// TIA Portal V17 export
// export: Created 2023-12-22T15:05:24.7176583Z, ExportSetting WithDefaults, DisplayName Totally Integrated Automation Portal, DisplayVersion V17, DisplayName TIA Portal Openness, DisplayVersion V17, DisplayName TIA Portal Version Control Interface, DisplayVersion V17, DisplayName STEP 7 Professional, DisplayVersion V17, DisplayName STEP 7 Safety, DisplayVersion V17, DisplayName WinCC Advanced, DisplayVersion V17
FUNCTION "Line_Alarms" : Void   // FC3, LAD
{ S7_Optimized_Access := 'TRUE' }
VERSION : 0.1
// stored: AutoNumber true, IsIECCheckEnabled false, SetENOAutomatically false, UDAEnableTagReadback false
   VAR_INPUT
      All_Lines : Int;   // Кол-во линий
   END_VAR
   VAR_IN_OUT
      Alm_REQ : Int;   // Запрос аварии
      Alm_Now : Int;   // Авария сейчас
      Ready : Bool;   // Готовность
   END_VAR
   VAR_TEMP   // added for the SCL form of the ladder/FBD networks
      _w1 : Bool;
      _w2 : Bool;
      _w3 : Bool;
      _w4 : Bool;
      _w5 : Bool;
      _w6 : Bool;
      _w7 : Bool;
   END_VAR
BEGIN

REGION Network 1: Проверка корректности выбранной линии
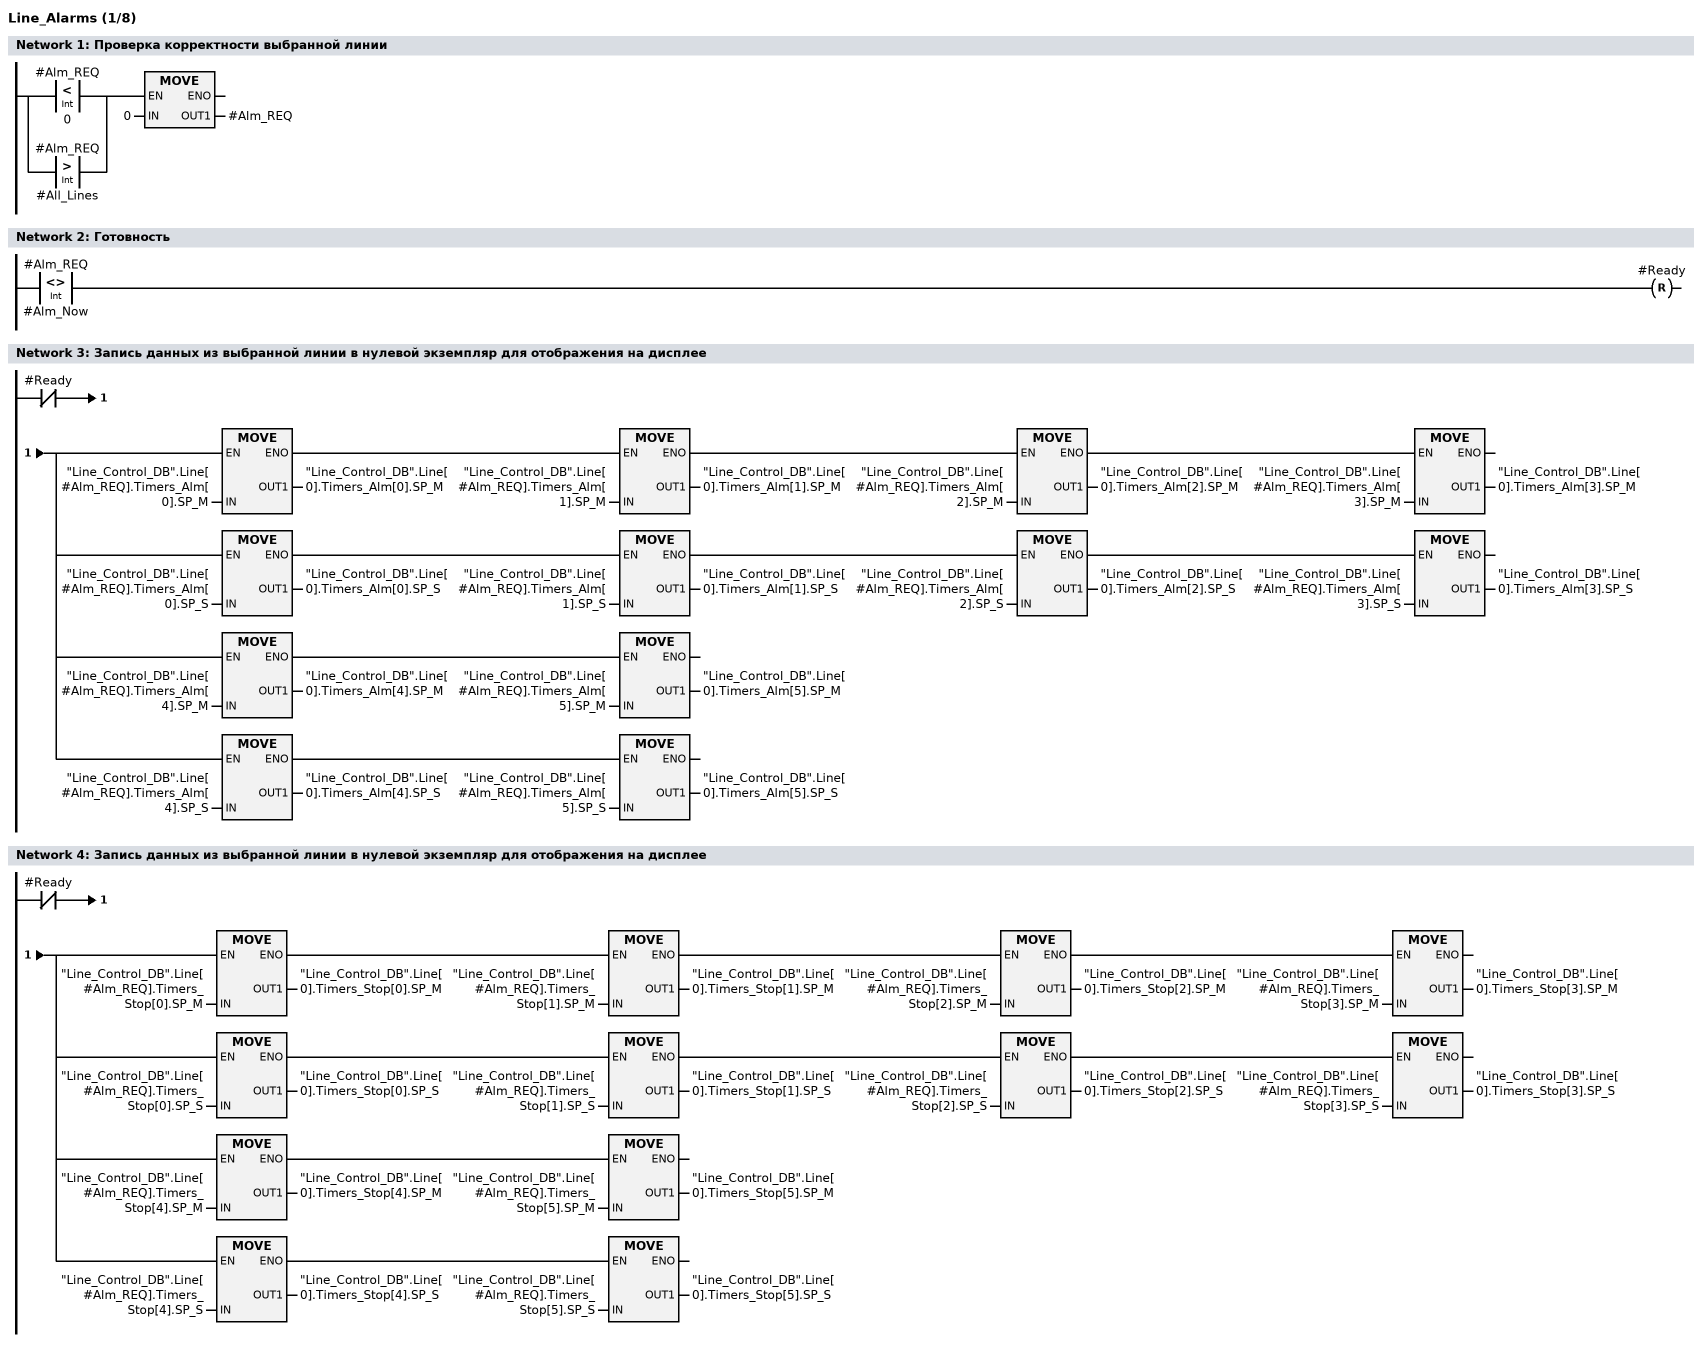
   RUNG wire#powerrail
      { S7_Templates := "SrcType := Int" } LT_Contact(in1 := #Alm_REQ, in2 := 0)
      wire#w1
      Move(in := 0, out1 => #Alm_REQ)
   END_RUNG
   RUNG wire#powerrail
      { S7_Templates := "SrcType := Int" } GT_Contact(in1 := #Alm_REQ, in2 := #All_Lines)
   END_RUNG wire#w1
   // the same network as SCL:
   IF (#Alm_REQ < 0) OR (#Alm_REQ > #All_Lines) THEN #Alm_REQ := 0; END_IF;
END_REGION

REGION Network 2: Готовность
   RUNG wire#powerrail
      { S7_Templates := "SrcType := Int" } NE_Contact(in1 := #Alm_REQ, in2 := #Alm_Now)
      R_Coil( #Ready )
   END_RUNG
   // the same network as SCL:
   IF #Alm_REQ <> #Alm_Now THEN #Ready := FALSE; END_IF;
END_REGION

REGION Network 3: Запись данных из выбранной линии в нулевой экземпляр для отображения на дисплее
   RUNG wire#powerrail
      I_Contact( #Ready )
      wire#w1
      Move(in := "Line_Control_DB".Line[#Alm_REQ].Timers_Alm[0].SP_M, out1 => "Line_Control_DB".Line[0].Timers_Alm[0].SP_M)
      Move(in := "Line_Control_DB".Line[#Alm_REQ].Timers_Alm[1].SP_M, out1 => "Line_Control_DB".Line[0].Timers_Alm[1].SP_M)
      Move(in := "Line_Control_DB".Line[#Alm_REQ].Timers_Alm[2].SP_M, out1 => "Line_Control_DB".Line[0].Timers_Alm[2].SP_M)
      Move(in := "Line_Control_DB".Line[#Alm_REQ].Timers_Alm[3].SP_M, out1 => "Line_Control_DB".Line[0].Timers_Alm[3].SP_M)
   END_RUNG
   RUNG wire#w1
      Move(in := "Line_Control_DB".Line[#Alm_REQ].Timers_Alm[0].SP_S, out1 => "Line_Control_DB".Line[0].Timers_Alm[0].SP_S)
      Move(in := "Line_Control_DB".Line[#Alm_REQ].Timers_Alm[1].SP_S, out1 => "Line_Control_DB".Line[0].Timers_Alm[1].SP_S)
      Move(in := "Line_Control_DB".Line[#Alm_REQ].Timers_Alm[2].SP_S, out1 => "Line_Control_DB".Line[0].Timers_Alm[2].SP_S)
      Move(in := "Line_Control_DB".Line[#Alm_REQ].Timers_Alm[3].SP_S, out1 => "Line_Control_DB".Line[0].Timers_Alm[3].SP_S)
   END_RUNG
   RUNG wire#w1
      Move(in := "Line_Control_DB".Line[#Alm_REQ].Timers_Alm[4].SP_M, out1 => "Line_Control_DB".Line[0].Timers_Alm[4].SP_M)
      Move(in := "Line_Control_DB".Line[#Alm_REQ].Timers_Alm[5].SP_M, out1 => "Line_Control_DB".Line[0].Timers_Alm[5].SP_M)
   END_RUNG
   RUNG wire#w1
      Move(in := "Line_Control_DB".Line[#Alm_REQ].Timers_Alm[4].SP_S, out1 => "Line_Control_DB".Line[0].Timers_Alm[4].SP_S)
      Move(in := "Line_Control_DB".Line[#Alm_REQ].Timers_Alm[5].SP_S, out1 => "Line_Control_DB".Line[0].Timers_Alm[5].SP_S)
   END_RUNG
   // the same network as SCL:
   IF NOT #Ready THEN
       "Line_Control_DB".Line[0].Timers_Alm[0].SP_M := "Line_Control_DB".Line[#Alm_REQ].Timers_Alm[0].SP_M;
       "Line_Control_DB".Line[0].Timers_Alm[1].SP_M := "Line_Control_DB".Line[#Alm_REQ].Timers_Alm[1].SP_M;
       "Line_Control_DB".Line[0].Timers_Alm[2].SP_M := "Line_Control_DB".Line[#Alm_REQ].Timers_Alm[2].SP_M;
       "Line_Control_DB".Line[0].Timers_Alm[3].SP_M := "Line_Control_DB".Line[#Alm_REQ].Timers_Alm[3].SP_M;
       "Line_Control_DB".Line[0].Timers_Alm[0].SP_S := "Line_Control_DB".Line[#Alm_REQ].Timers_Alm[0].SP_S;
       "Line_Control_DB".Line[0].Timers_Alm[1].SP_S := "Line_Control_DB".Line[#Alm_REQ].Timers_Alm[1].SP_S;
       "Line_Control_DB".Line[0].Timers_Alm[2].SP_S := "Line_Control_DB".Line[#Alm_REQ].Timers_Alm[2].SP_S;
       "Line_Control_DB".Line[0].Timers_Alm[3].SP_S := "Line_Control_DB".Line[#Alm_REQ].Timers_Alm[3].SP_S;
       "Line_Control_DB".Line[0].Timers_Alm[4].SP_M := "Line_Control_DB".Line[#Alm_REQ].Timers_Alm[4].SP_M;
       "Line_Control_DB".Line[0].Timers_Alm[5].SP_M := "Line_Control_DB".Line[#Alm_REQ].Timers_Alm[5].SP_M;
       "Line_Control_DB".Line[0].Timers_Alm[4].SP_S := "Line_Control_DB".Line[#Alm_REQ].Timers_Alm[4].SP_S;
       "Line_Control_DB".Line[0].Timers_Alm[5].SP_S := "Line_Control_DB".Line[#Alm_REQ].Timers_Alm[5].SP_S;
   END_IF;
END_REGION

REGION Network 4: Запись данных из выбранной линии в нулевой экземпляр для отображения на дисплее
   RUNG wire#powerrail
      I_Contact( #Ready )
      wire#w1
      Move(in := "Line_Control_DB".Line[#Alm_REQ].Timers_Stop[0].SP_M, out1 => "Line_Control_DB".Line[0].Timers_Stop[0].SP_M)
      Move(in := "Line_Control_DB".Line[#Alm_REQ].Timers_Stop[1].SP_M, out1 => "Line_Control_DB".Line[0].Timers_Stop[1].SP_M)
      Move(in := "Line_Control_DB".Line[#Alm_REQ].Timers_Stop[2].SP_M, out1 => "Line_Control_DB".Line[0].Timers_Stop[2].SP_M)
      Move(in := "Line_Control_DB".Line[#Alm_REQ].Timers_Stop[3].SP_M, out1 => "Line_Control_DB".Line[0].Timers_Stop[3].SP_M)
   END_RUNG
   RUNG wire#w1
      Move(in := "Line_Control_DB".Line[#Alm_REQ].Timers_Stop[0].SP_S, out1 => "Line_Control_DB".Line[0].Timers_Stop[0].SP_S)
      Move(in := "Line_Control_DB".Line[#Alm_REQ].Timers_Stop[1].SP_S, out1 => "Line_Control_DB".Line[0].Timers_Stop[1].SP_S)
      Move(in := "Line_Control_DB".Line[#Alm_REQ].Timers_Stop[2].SP_S, out1 => "Line_Control_DB".Line[0].Timers_Stop[2].SP_S)
      Move(in := "Line_Control_DB".Line[#Alm_REQ].Timers_Stop[3].SP_S, out1 => "Line_Control_DB".Line[0].Timers_Stop[3].SP_S)
   END_RUNG
   RUNG wire#w1
      Move(in := "Line_Control_DB".Line[#Alm_REQ].Timers_Stop[4].SP_M, out1 => "Line_Control_DB".Line[0].Timers_Stop[4].SP_M)
      Move(in := "Line_Control_DB".Line[#Alm_REQ].Timers_Stop[5].SP_M, out1 => "Line_Control_DB".Line[0].Timers_Stop[5].SP_M)
   END_RUNG
   RUNG wire#w1
      Move(in := "Line_Control_DB".Line[#Alm_REQ].Timers_Stop[4].SP_S, out1 => "Line_Control_DB".Line[0].Timers_Stop[4].SP_S)
      Move(in := "Line_Control_DB".Line[#Alm_REQ].Timers_Stop[5].SP_S, out1 => "Line_Control_DB".Line[0].Timers_Stop[5].SP_S)
   END_RUNG
   // the same network as SCL:
   IF NOT #Ready THEN
       "Line_Control_DB".Line[0].Timers_Stop[0].SP_M := "Line_Control_DB".Line[#Alm_REQ].Timers_Stop[0].SP_M;
       "Line_Control_DB".Line[0].Timers_Stop[1].SP_M := "Line_Control_DB".Line[#Alm_REQ].Timers_Stop[1].SP_M;
       "Line_Control_DB".Line[0].Timers_Stop[2].SP_M := "Line_Control_DB".Line[#Alm_REQ].Timers_Stop[2].SP_M;
       "Line_Control_DB".Line[0].Timers_Stop[3].SP_M := "Line_Control_DB".Line[#Alm_REQ].Timers_Stop[3].SP_M;
       "Line_Control_DB".Line[0].Timers_Stop[0].SP_S := "Line_Control_DB".Line[#Alm_REQ].Timers_Stop[0].SP_S;
       "Line_Control_DB".Line[0].Timers_Stop[1].SP_S := "Line_Control_DB".Line[#Alm_REQ].Timers_Stop[1].SP_S;
       "Line_Control_DB".Line[0].Timers_Stop[2].SP_S := "Line_Control_DB".Line[#Alm_REQ].Timers_Stop[2].SP_S;
       "Line_Control_DB".Line[0].Timers_Stop[3].SP_S := "Line_Control_DB".Line[#Alm_REQ].Timers_Stop[3].SP_S;
       "Line_Control_DB".Line[0].Timers_Stop[4].SP_M := "Line_Control_DB".Line[#Alm_REQ].Timers_Stop[4].SP_M;
       "Line_Control_DB".Line[0].Timers_Stop[5].SP_M := "Line_Control_DB".Line[#Alm_REQ].Timers_Stop[5].SP_M;
       "Line_Control_DB".Line[0].Timers_Stop[4].SP_S := "Line_Control_DB".Line[#Alm_REQ].Timers_Stop[4].SP_S;
       "Line_Control_DB".Line[0].Timers_Stop[5].SP_S := "Line_Control_DB".Line[#Alm_REQ].Timers_Stop[5].SP_S;
   END_IF;
END_REGION

REGION Network 5: Запись данных из выбранной линии в нулевой экземпляр для отображения на дисплее
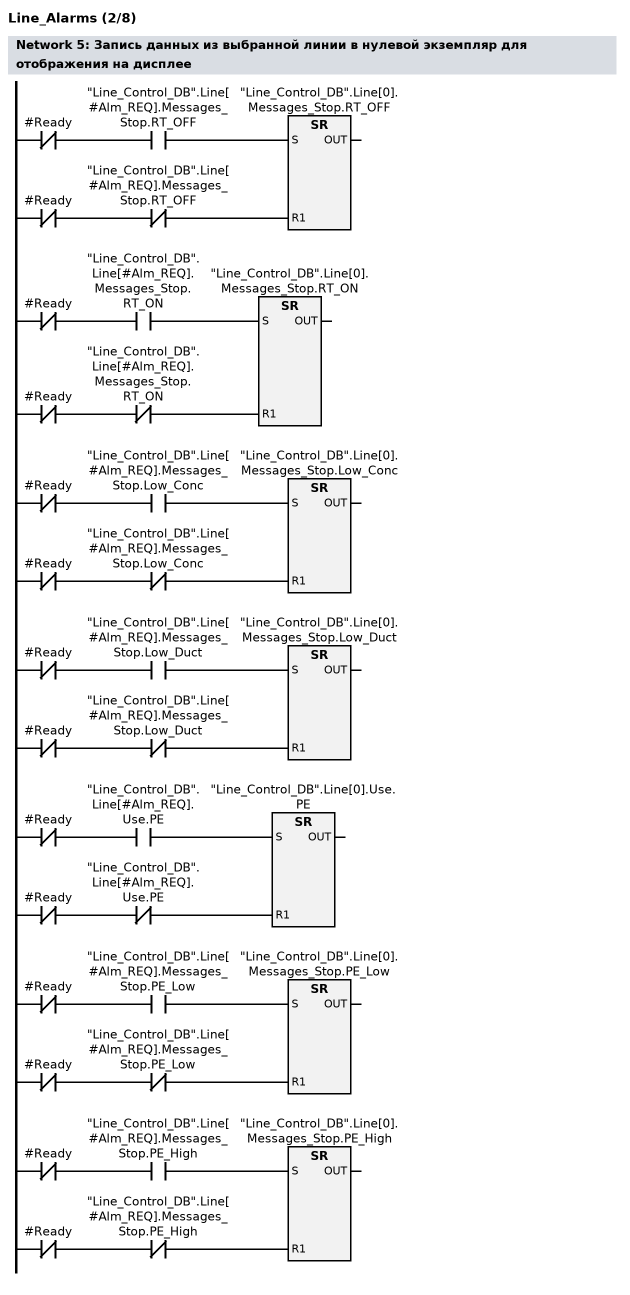
   RUNG wire#powerrail
      I_Contact( #Ready )
      Contact( "Line_Control_DB".Line[#Alm_REQ].Messages_Stop.RT_OFF )
      S_SR(operand := "Line_Control_DB".Line[0].Messages_Stop.RT_OFF, r1 := wire#w1)
   END_RUNG
   RUNG wire#powerrail
      I_Contact( #Ready )
      I_Contact( "Line_Control_DB".Line[#Alm_REQ].Messages_Stop.RT_OFF )
   END_RUNG wire#w1
   RUNG wire#powerrail
      I_Contact( #Ready )
      Contact( "Line_Control_DB".Line[#Alm_REQ].Messages_Stop.RT_ON )
      S_SR(operand := "Line_Control_DB".Line[0].Messages_Stop.RT_ON, r1 := wire#w2)
   END_RUNG
   RUNG wire#powerrail
      I_Contact( #Ready )
      I_Contact( "Line_Control_DB".Line[#Alm_REQ].Messages_Stop.RT_ON )
   END_RUNG wire#w2
   RUNG wire#powerrail
      I_Contact( #Ready )
      Contact( "Line_Control_DB".Line[#Alm_REQ].Messages_Stop.Low_Conc )
      S_SR(operand := "Line_Control_DB".Line[0].Messages_Stop.Low_Conc, r1 := wire#w3)
   END_RUNG
   RUNG wire#powerrail
      I_Contact( #Ready )
      I_Contact( "Line_Control_DB".Line[#Alm_REQ].Messages_Stop.Low_Conc )
   END_RUNG wire#w3
   RUNG wire#powerrail
      I_Contact( #Ready )
      Contact( "Line_Control_DB".Line[#Alm_REQ].Messages_Stop.Low_Duct )
      S_SR(operand := "Line_Control_DB".Line[0].Messages_Stop.Low_Duct, r1 := wire#w4)
   END_RUNG
   RUNG wire#powerrail
      I_Contact( #Ready )
      I_Contact( "Line_Control_DB".Line[#Alm_REQ].Messages_Stop.Low_Duct )
   END_RUNG wire#w4
   RUNG wire#powerrail
      I_Contact( #Ready )
      Contact( "Line_Control_DB".Line[#Alm_REQ].Use.PE )
      S_SR(operand := "Line_Control_DB".Line[0].Use.PE, r1 := wire#w5)
   END_RUNG
   RUNG wire#powerrail
      I_Contact( #Ready )
      I_Contact( "Line_Control_DB".Line[#Alm_REQ].Use.PE )
   END_RUNG wire#w5
   RUNG wire#powerrail
      I_Contact( #Ready )
      Contact( "Line_Control_DB".Line[#Alm_REQ].Messages_Stop.PE_Low )
      S_SR(operand := "Line_Control_DB".Line[0].Messages_Stop.PE_Low, r1 := wire#w6)
   END_RUNG
   RUNG wire#powerrail
      I_Contact( #Ready )
      I_Contact( "Line_Control_DB".Line[#Alm_REQ].Messages_Stop.PE_Low )
   END_RUNG wire#w6
   RUNG wire#powerrail
      I_Contact( #Ready )
      Contact( "Line_Control_DB".Line[#Alm_REQ].Messages_Stop.PE_High )
      S_SR(operand := "Line_Control_DB".Line[0].Messages_Stop.PE_High, r1 := wire#w7)
   END_RUNG
   RUNG wire#powerrail
      I_Contact( #Ready )
      I_Contact( "Line_Control_DB".Line[#Alm_REQ].Messages_Stop.PE_High )
   END_RUNG wire#w7
   // the same network as SCL:
   #_w1 := NOT #Ready AND NOT "Line_Control_DB".Line[#Alm_REQ].Messages_Stop.RT_OFF;
   IF NOT #Ready AND "Line_Control_DB".Line[#Alm_REQ].Messages_Stop.RT_OFF THEN
       "Line_Control_DB".Line[0].Messages_Stop.RT_OFF := TRUE;   // SR flip-flop
   END_IF;
   IF #_w1 THEN "Line_Control_DB".Line[0].Messages_Stop.RT_OFF := FALSE; END_IF;
   #_w2 := NOT #Ready AND NOT "Line_Control_DB".Line[#Alm_REQ].Messages_Stop.RT_ON;
   IF NOT #Ready AND "Line_Control_DB".Line[#Alm_REQ].Messages_Stop.RT_ON THEN
       "Line_Control_DB".Line[0].Messages_Stop.RT_ON := TRUE;   // SR flip-flop
   END_IF;
   IF #_w2 THEN "Line_Control_DB".Line[0].Messages_Stop.RT_ON := FALSE; END_IF;
   #_w3 := NOT #Ready AND NOT "Line_Control_DB".Line[#Alm_REQ].Messages_Stop.Low_Conc;
   IF NOT #Ready AND "Line_Control_DB".Line[#Alm_REQ].Messages_Stop.Low_Conc THEN
       "Line_Control_DB".Line[0].Messages_Stop.Low_Conc := TRUE;   // SR flip-flop
   END_IF;
   IF #_w3 THEN "Line_Control_DB".Line[0].Messages_Stop.Low_Conc := FALSE; END_IF;
   #_w4 := NOT #Ready AND NOT "Line_Control_DB".Line[#Alm_REQ].Messages_Stop.Low_Duct;
   IF NOT #Ready AND "Line_Control_DB".Line[#Alm_REQ].Messages_Stop.Low_Duct THEN
       "Line_Control_DB".Line[0].Messages_Stop.Low_Duct := TRUE;   // SR flip-flop
   END_IF;
   IF #_w4 THEN "Line_Control_DB".Line[0].Messages_Stop.Low_Duct := FALSE; END_IF;
   #_w5 := NOT #Ready AND NOT "Line_Control_DB".Line[#Alm_REQ].Use.PE;
   IF NOT #Ready AND "Line_Control_DB".Line[#Alm_REQ].Use.PE THEN
       "Line_Control_DB".Line[0].Use.PE := TRUE;   // SR flip-flop
   END_IF;
   IF #_w5 THEN "Line_Control_DB".Line[0].Use.PE := FALSE; END_IF;
   #_w6 := NOT #Ready AND NOT "Line_Control_DB".Line[#Alm_REQ].Messages_Stop.PE_Low;
   IF NOT #Ready AND "Line_Control_DB".Line[#Alm_REQ].Messages_Stop.PE_Low THEN
       "Line_Control_DB".Line[0].Messages_Stop.PE_Low := TRUE;   // SR flip-flop
   END_IF;
   IF #_w6 THEN "Line_Control_DB".Line[0].Messages_Stop.PE_Low := FALSE; END_IF;
   #_w7 := NOT #Ready AND NOT "Line_Control_DB".Line[#Alm_REQ].Messages_Stop.PE_High;
   IF NOT #Ready AND "Line_Control_DB".Line[#Alm_REQ].Messages_Stop.PE_High THEN
       "Line_Control_DB".Line[0].Messages_Stop.PE_High := TRUE;   // SR flip-flop
   END_IF;
   IF #_w7 THEN "Line_Control_DB".Line[0].Messages_Stop.PE_High := FALSE; END_IF;
END_REGION

REGION Network 6: Запись данных из выбранной линии в нулевой экземпляр для отображения на дисплее
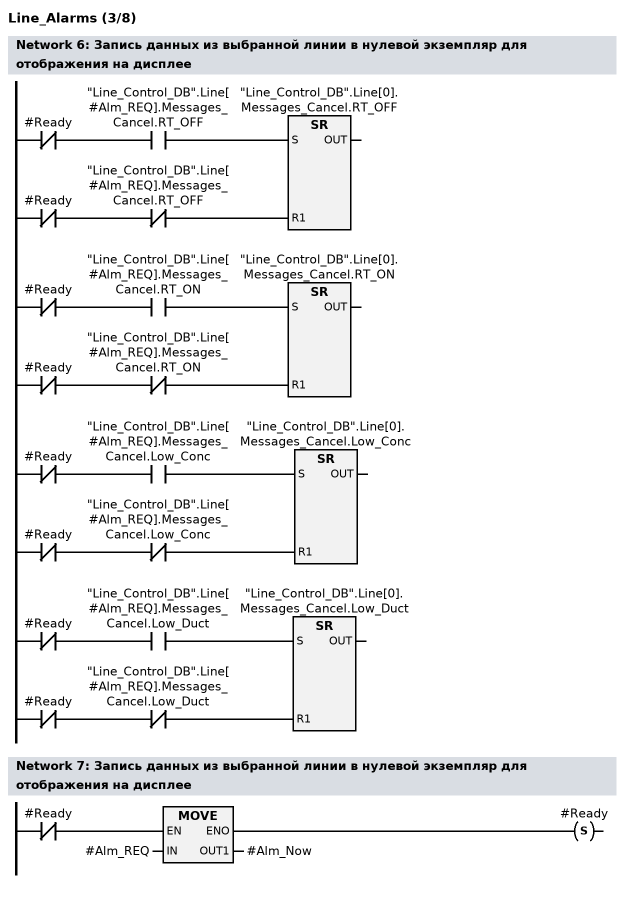
   RUNG wire#powerrail
      I_Contact( #Ready )
      Contact( "Line_Control_DB".Line[#Alm_REQ].Messages_Cancel.RT_OFF )
      S_SR(operand := "Line_Control_DB".Line[0].Messages_Cancel.RT_OFF, r1 := wire#w1)
   END_RUNG
   RUNG wire#powerrail
      I_Contact( #Ready )
      I_Contact( "Line_Control_DB".Line[#Alm_REQ].Messages_Cancel.RT_OFF )
   END_RUNG wire#w1
   RUNG wire#powerrail
      I_Contact( #Ready )
      Contact( "Line_Control_DB".Line[#Alm_REQ].Messages_Cancel.RT_ON )
      S_SR(operand := "Line_Control_DB".Line[0].Messages_Cancel.RT_ON, r1 := wire#w2)
   END_RUNG
   RUNG wire#powerrail
      I_Contact( #Ready )
      I_Contact( "Line_Control_DB".Line[#Alm_REQ].Messages_Cancel.RT_ON )
   END_RUNG wire#w2
   RUNG wire#powerrail
      I_Contact( #Ready )
      Contact( "Line_Control_DB".Line[#Alm_REQ].Messages_Cancel.Low_Conc )
      S_SR(operand := "Line_Control_DB".Line[0].Messages_Cancel.Low_Conc, r1 := wire#w3)
   END_RUNG
   RUNG wire#powerrail
      I_Contact( #Ready )
      I_Contact( "Line_Control_DB".Line[#Alm_REQ].Messages_Cancel.Low_Conc )
   END_RUNG wire#w3
   RUNG wire#powerrail
      I_Contact( #Ready )
      Contact( "Line_Control_DB".Line[#Alm_REQ].Messages_Cancel.Low_Duct )
      S_SR(operand := "Line_Control_DB".Line[0].Messages_Cancel.Low_Duct, r1 := wire#w4)
   END_RUNG
   RUNG wire#powerrail
      I_Contact( #Ready )
      I_Contact( "Line_Control_DB".Line[#Alm_REQ].Messages_Cancel.Low_Duct )
   END_RUNG wire#w4
   // the same network as SCL:
   #_w1 := NOT #Ready AND NOT "Line_Control_DB".Line[#Alm_REQ].Messages_Cancel.RT_OFF;
   IF NOT #Ready AND "Line_Control_DB".Line[#Alm_REQ].Messages_Cancel.RT_OFF THEN
       "Line_Control_DB".Line[0].Messages_Cancel.RT_OFF := TRUE;   // SR flip-flop
   END_IF;
   IF #_w1 THEN "Line_Control_DB".Line[0].Messages_Cancel.RT_OFF := FALSE; END_IF;
   #_w2 := NOT #Ready AND NOT "Line_Control_DB".Line[#Alm_REQ].Messages_Cancel.RT_ON;
   IF NOT #Ready AND "Line_Control_DB".Line[#Alm_REQ].Messages_Cancel.RT_ON THEN
       "Line_Control_DB".Line[0].Messages_Cancel.RT_ON := TRUE;   // SR flip-flop
   END_IF;
   IF #_w2 THEN "Line_Control_DB".Line[0].Messages_Cancel.RT_ON := FALSE; END_IF;
   #_w3 := NOT #Ready AND NOT "Line_Control_DB".Line[#Alm_REQ].Messages_Cancel.Low_Conc;
   IF NOT #Ready AND "Line_Control_DB".Line[#Alm_REQ].Messages_Cancel.Low_Conc THEN
       "Line_Control_DB".Line[0].Messages_Cancel.Low_Conc := TRUE;   // SR flip-flop
   END_IF;
   IF #_w3 THEN "Line_Control_DB".Line[0].Messages_Cancel.Low_Conc := FALSE; END_IF;
   #_w4 := NOT #Ready AND NOT "Line_Control_DB".Line[#Alm_REQ].Messages_Cancel.Low_Duct;
   IF NOT #Ready AND "Line_Control_DB".Line[#Alm_REQ].Messages_Cancel.Low_Duct THEN
       "Line_Control_DB".Line[0].Messages_Cancel.Low_Duct := TRUE;   // SR flip-flop
   END_IF;
   IF #_w4 THEN "Line_Control_DB".Line[0].Messages_Cancel.Low_Duct := FALSE; END_IF;
END_REGION

REGION Network 7: Запись данных из выбранной линии в нулевой экземпляр для отображения на дисплее
   RUNG wire#powerrail
      I_Contact( #Ready )
      Move(in := #Alm_REQ, out1 => #Alm_Now)
      S_Coil( #Ready )
   END_RUNG
   // the same network as SCL:
   IF NOT #Ready THEN
       #Alm_Now := #Alm_REQ;
       #Ready := TRUE;
   END_IF;
END_REGION

REGION Network 8: Запись данных из выбранной линии в нулевой экземпляр для отображения на дисплее
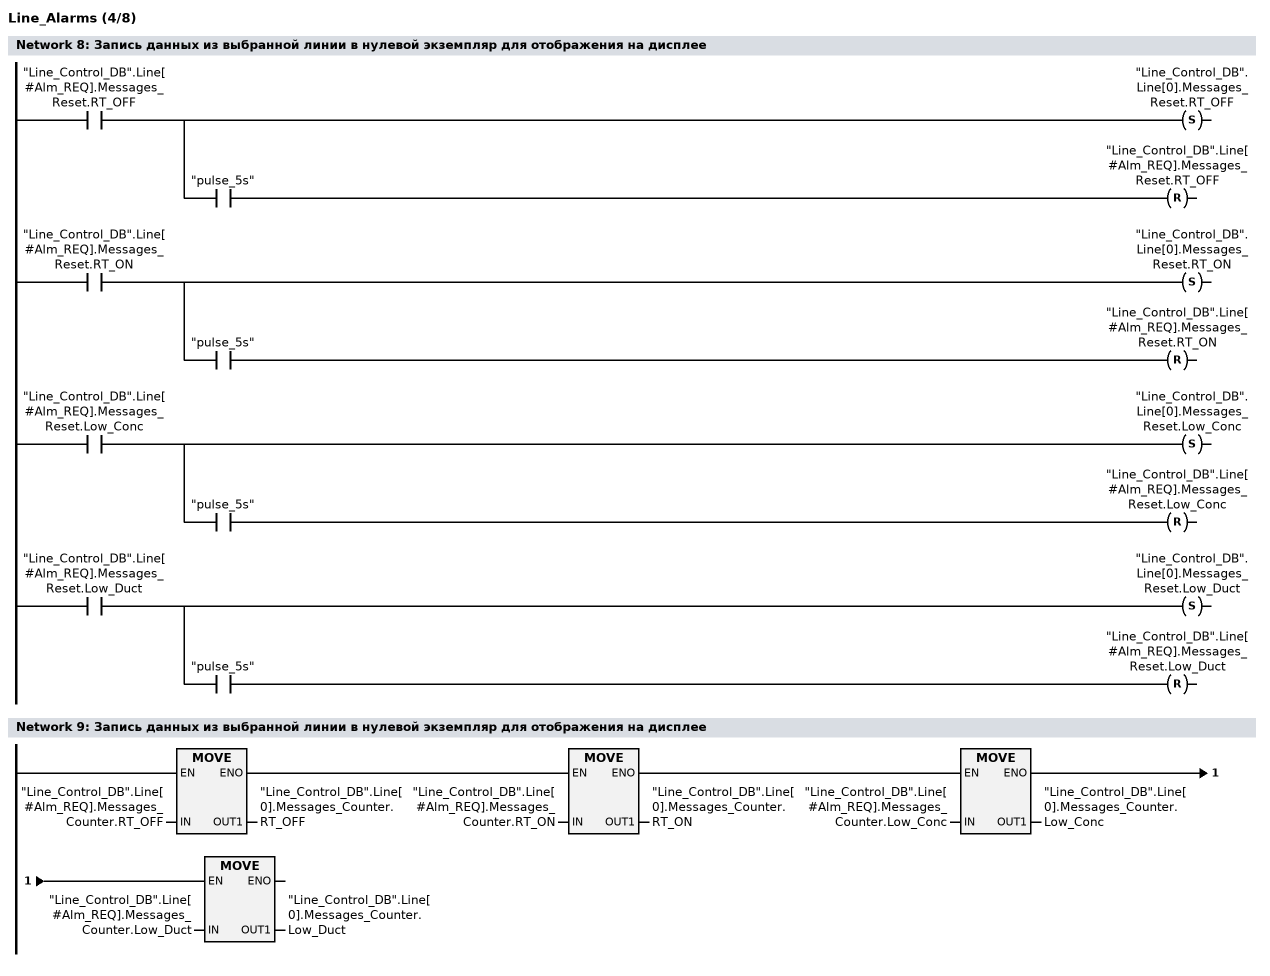
   RUNG wire#powerrail
      Contact( "Line_Control_DB".Line[#Alm_REQ].Messages_Reset.RT_OFF )
      wire#w1
      S_Coil( "Line_Control_DB".Line[0].Messages_Reset.RT_OFF )
   END_RUNG
   RUNG wire#w1
      Contact( "pulse_5s" )
      R_Coil( "Line_Control_DB".Line[#Alm_REQ].Messages_Reset.RT_OFF )
   END_RUNG
   RUNG wire#powerrail
      Contact( "Line_Control_DB".Line[#Alm_REQ].Messages_Reset.RT_ON )
      wire#w2
      S_Coil( "Line_Control_DB".Line[0].Messages_Reset.RT_ON )
   END_RUNG
   RUNG wire#w2
      Contact( "pulse_5s" )
      R_Coil( "Line_Control_DB".Line[#Alm_REQ].Messages_Reset.RT_ON )
   END_RUNG
   RUNG wire#powerrail
      Contact( "Line_Control_DB".Line[#Alm_REQ].Messages_Reset.Low_Conc )
      wire#w3
      S_Coil( "Line_Control_DB".Line[0].Messages_Reset.Low_Conc )
   END_RUNG
   RUNG wire#w3
      Contact( "pulse_5s" )
      R_Coil( "Line_Control_DB".Line[#Alm_REQ].Messages_Reset.Low_Conc )
   END_RUNG
   RUNG wire#powerrail
      Contact( "Line_Control_DB".Line[#Alm_REQ].Messages_Reset.Low_Duct )
      wire#w4
      S_Coil( "Line_Control_DB".Line[0].Messages_Reset.Low_Duct )
   END_RUNG
   RUNG wire#w4
      Contact( "pulse_5s" )
      R_Coil( "Line_Control_DB".Line[#Alm_REQ].Messages_Reset.Low_Duct )
   END_RUNG
   // the same network as SCL:
   #_w1 := "Line_Control_DB".Line[#Alm_REQ].Messages_Reset.RT_OFF;
   IF #_w1 THEN "Line_Control_DB".Line[0].Messages_Reset.RT_OFF := TRUE; END_IF;
   IF #_w1 AND "pulse_5s" THEN "Line_Control_DB".Line[#Alm_REQ].Messages_Reset.RT_OFF := FALSE; END_IF;
   #_w2 := "Line_Control_DB".Line[#Alm_REQ].Messages_Reset.RT_ON;
   IF #_w2 THEN "Line_Control_DB".Line[0].Messages_Reset.RT_ON := TRUE; END_IF;
   IF #_w2 AND "pulse_5s" THEN "Line_Control_DB".Line[#Alm_REQ].Messages_Reset.RT_ON := FALSE; END_IF;
   #_w3 := "Line_Control_DB".Line[#Alm_REQ].Messages_Reset.Low_Conc;
   IF #_w3 THEN "Line_Control_DB".Line[0].Messages_Reset.Low_Conc := TRUE; END_IF;
   IF #_w3 AND "pulse_5s" THEN "Line_Control_DB".Line[#Alm_REQ].Messages_Reset.Low_Conc := FALSE; END_IF;
   #_w4 := "Line_Control_DB".Line[#Alm_REQ].Messages_Reset.Low_Duct;
   IF #_w4 THEN "Line_Control_DB".Line[0].Messages_Reset.Low_Duct := TRUE; END_IF;
   IF #_w4 AND "pulse_5s" THEN "Line_Control_DB".Line[#Alm_REQ].Messages_Reset.Low_Duct := FALSE; END_IF;
END_REGION

REGION Network 9: Запись данных из выбранной линии в нулевой экземпляр для отображения на дисплее
   RUNG wire#powerrail
      Move(in := "Line_Control_DB".Line[#Alm_REQ].Messages_Counter.RT_OFF, out1 => "Line_Control_DB".Line[0].Messages_Counter.RT_OFF)
      Move(in := "Line_Control_DB".Line[#Alm_REQ].Messages_Counter.RT_ON, out1 => "Line_Control_DB".Line[0].Messages_Counter.RT_ON)
      Move(in := "Line_Control_DB".Line[#Alm_REQ].Messages_Counter.Low_Conc, out1 => "Line_Control_DB".Line[0].Messages_Counter.Low_Conc)
      Move(in := "Line_Control_DB".Line[#Alm_REQ].Messages_Counter.Low_Duct, out1 => "Line_Control_DB".Line[0].Messages_Counter.Low_Duct)
   END_RUNG
   // the same network as SCL:
   "Line_Control_DB".Line[0].Messages_Counter.RT_OFF := "Line_Control_DB".Line[#Alm_REQ].Messages_Counter.RT_OFF;
   "Line_Control_DB".Line[0].Messages_Counter.RT_ON := "Line_Control_DB".Line[#Alm_REQ].Messages_Counter.RT_ON;
   "Line_Control_DB".Line[0].Messages_Counter.Low_Conc := "Line_Control_DB".Line[#Alm_REQ].Messages_Counter.Low_Conc;
   "Line_Control_DB".Line[0].Messages_Counter.Low_Duct := "Line_Control_DB".Line[#Alm_REQ].Messages_Counter.Low_Duct;
END_REGION

REGION Network 10: Чтение данных из выбранной линии в нулевой экземпляр для отображения на дисплее
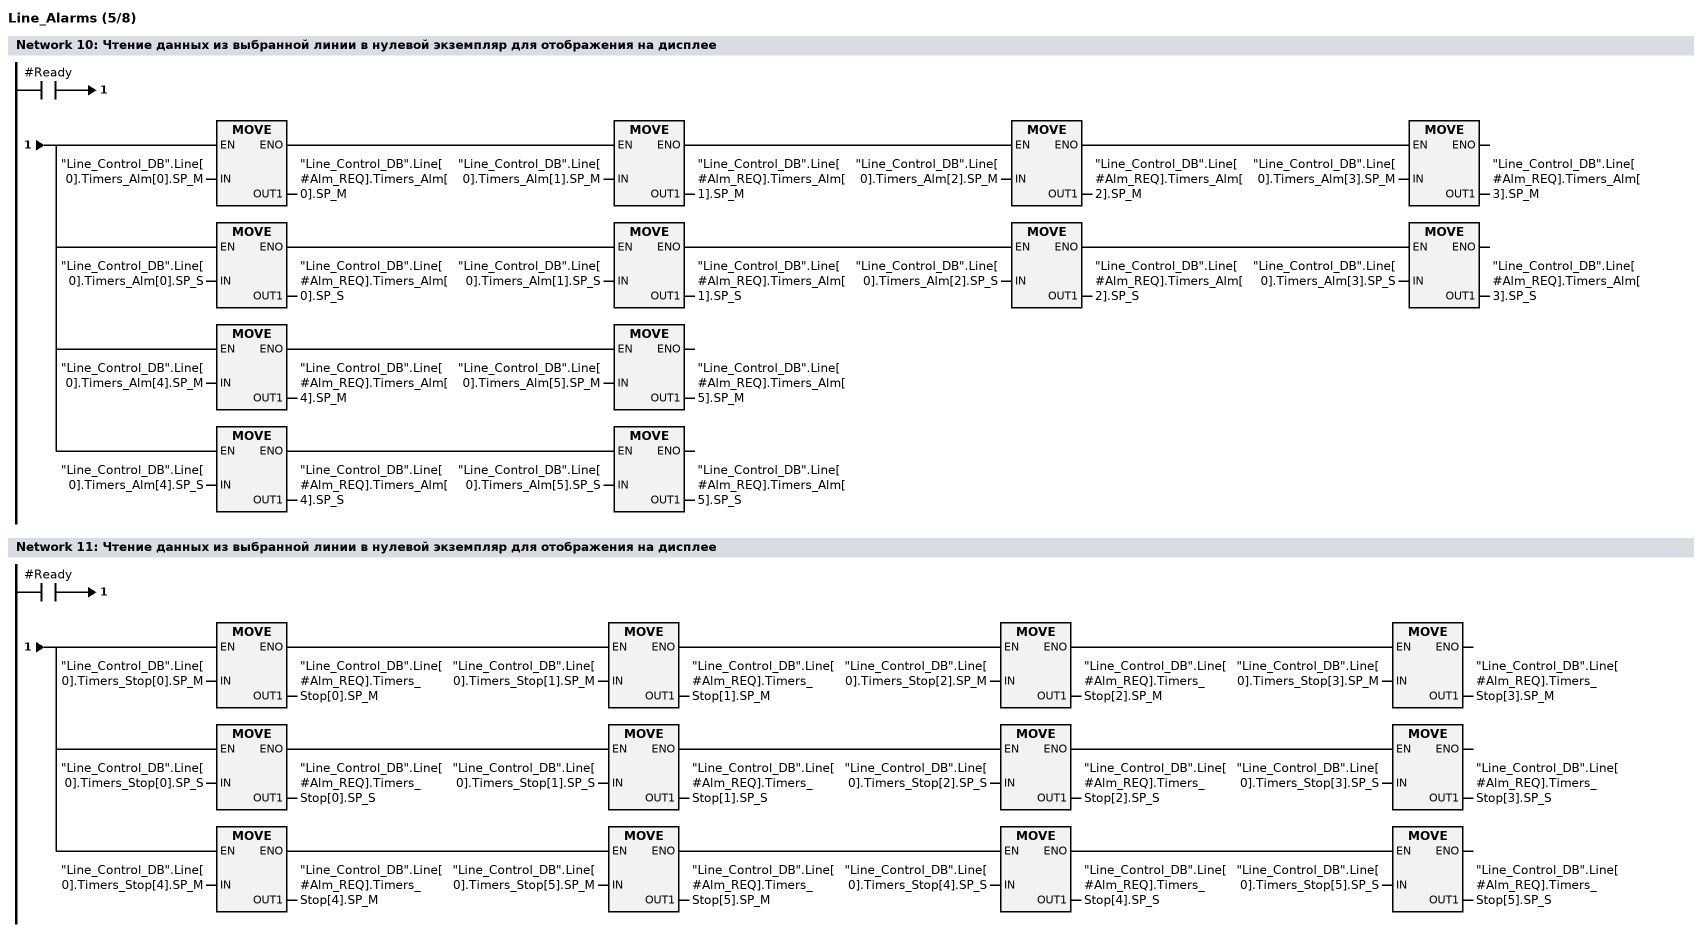
   RUNG wire#powerrail
      Contact( #Ready )
      wire#w1
      Move(in := "Line_Control_DB".Line[0].Timers_Alm[0].SP_M, out1 => "Line_Control_DB".Line[#Alm_REQ].Timers_Alm[0].SP_M)
      Move(in := "Line_Control_DB".Line[0].Timers_Alm[1].SP_M, out1 => "Line_Control_DB".Line[#Alm_REQ].Timers_Alm[1].SP_M)
      Move(in := "Line_Control_DB".Line[0].Timers_Alm[2].SP_M, out1 => "Line_Control_DB".Line[#Alm_REQ].Timers_Alm[2].SP_M)
      Move(in := "Line_Control_DB".Line[0].Timers_Alm[3].SP_M, out1 => "Line_Control_DB".Line[#Alm_REQ].Timers_Alm[3].SP_M)
   END_RUNG
   RUNG wire#w1
      Move(in := "Line_Control_DB".Line[0].Timers_Alm[0].SP_S, out1 => "Line_Control_DB".Line[#Alm_REQ].Timers_Alm[0].SP_S)
      Move(in := "Line_Control_DB".Line[0].Timers_Alm[1].SP_S, out1 => "Line_Control_DB".Line[#Alm_REQ].Timers_Alm[1].SP_S)
      Move(in := "Line_Control_DB".Line[0].Timers_Alm[2].SP_S, out1 => "Line_Control_DB".Line[#Alm_REQ].Timers_Alm[2].SP_S)
      Move(in := "Line_Control_DB".Line[0].Timers_Alm[3].SP_S, out1 => "Line_Control_DB".Line[#Alm_REQ].Timers_Alm[3].SP_S)
   END_RUNG
   RUNG wire#w1
      Move(in := "Line_Control_DB".Line[0].Timers_Alm[4].SP_M, out1 => "Line_Control_DB".Line[#Alm_REQ].Timers_Alm[4].SP_M)
      Move(in := "Line_Control_DB".Line[0].Timers_Alm[5].SP_M, out1 => "Line_Control_DB".Line[#Alm_REQ].Timers_Alm[5].SP_M)
   END_RUNG
   RUNG wire#w1
      Move(in := "Line_Control_DB".Line[0].Timers_Alm[4].SP_S, out1 => "Line_Control_DB".Line[#Alm_REQ].Timers_Alm[4].SP_S)
      Move(in := "Line_Control_DB".Line[0].Timers_Alm[5].SP_S, out1 => "Line_Control_DB".Line[#Alm_REQ].Timers_Alm[5].SP_S)
   END_RUNG
   // the same network as SCL:
   IF #Ready THEN
       "Line_Control_DB".Line[#Alm_REQ].Timers_Alm[0].SP_M := "Line_Control_DB".Line[0].Timers_Alm[0].SP_M;
       "Line_Control_DB".Line[#Alm_REQ].Timers_Alm[1].SP_M := "Line_Control_DB".Line[0].Timers_Alm[1].SP_M;
       "Line_Control_DB".Line[#Alm_REQ].Timers_Alm[2].SP_M := "Line_Control_DB".Line[0].Timers_Alm[2].SP_M;
       "Line_Control_DB".Line[#Alm_REQ].Timers_Alm[3].SP_M := "Line_Control_DB".Line[0].Timers_Alm[3].SP_M;
       "Line_Control_DB".Line[#Alm_REQ].Timers_Alm[0].SP_S := "Line_Control_DB".Line[0].Timers_Alm[0].SP_S;
       "Line_Control_DB".Line[#Alm_REQ].Timers_Alm[1].SP_S := "Line_Control_DB".Line[0].Timers_Alm[1].SP_S;
       "Line_Control_DB".Line[#Alm_REQ].Timers_Alm[2].SP_S := "Line_Control_DB".Line[0].Timers_Alm[2].SP_S;
       "Line_Control_DB".Line[#Alm_REQ].Timers_Alm[3].SP_S := "Line_Control_DB".Line[0].Timers_Alm[3].SP_S;
       "Line_Control_DB".Line[#Alm_REQ].Timers_Alm[4].SP_M := "Line_Control_DB".Line[0].Timers_Alm[4].SP_M;
       "Line_Control_DB".Line[#Alm_REQ].Timers_Alm[5].SP_M := "Line_Control_DB".Line[0].Timers_Alm[5].SP_M;
       "Line_Control_DB".Line[#Alm_REQ].Timers_Alm[4].SP_S := "Line_Control_DB".Line[0].Timers_Alm[4].SP_S;
       "Line_Control_DB".Line[#Alm_REQ].Timers_Alm[5].SP_S := "Line_Control_DB".Line[0].Timers_Alm[5].SP_S;
   END_IF;
END_REGION

REGION Network 11: Чтение данных из выбранной линии в нулевой экземпляр для отображения на дисплее
   RUNG wire#powerrail
      Contact( #Ready )
      wire#w1
      Move(in := "Line_Control_DB".Line[0].Timers_Stop[0].SP_M, out1 => "Line_Control_DB".Line[#Alm_REQ].Timers_Stop[0].SP_M)
      Move(in := "Line_Control_DB".Line[0].Timers_Stop[1].SP_M, out1 => "Line_Control_DB".Line[#Alm_REQ].Timers_Stop[1].SP_M)
      Move(in := "Line_Control_DB".Line[0].Timers_Stop[2].SP_M, out1 => "Line_Control_DB".Line[#Alm_REQ].Timers_Stop[2].SP_M)
      Move(in := "Line_Control_DB".Line[0].Timers_Stop[3].SP_M, out1 => "Line_Control_DB".Line[#Alm_REQ].Timers_Stop[3].SP_M)
   END_RUNG
   RUNG wire#w1
      Move(in := "Line_Control_DB".Line[0].Timers_Stop[0].SP_S, out1 => "Line_Control_DB".Line[#Alm_REQ].Timers_Stop[0].SP_S)
      Move(in := "Line_Control_DB".Line[0].Timers_Stop[1].SP_S, out1 => "Line_Control_DB".Line[#Alm_REQ].Timers_Stop[1].SP_S)
      Move(in := "Line_Control_DB".Line[0].Timers_Stop[2].SP_S, out1 => "Line_Control_DB".Line[#Alm_REQ].Timers_Stop[2].SP_S)
      Move(in := "Line_Control_DB".Line[0].Timers_Stop[3].SP_S, out1 => "Line_Control_DB".Line[#Alm_REQ].Timers_Stop[3].SP_S)
   END_RUNG
   RUNG wire#w1
      Move(in := "Line_Control_DB".Line[0].Timers_Stop[4].SP_M, out1 => "Line_Control_DB".Line[#Alm_REQ].Timers_Stop[4].SP_M)
      Move(in := "Line_Control_DB".Line[0].Timers_Stop[5].SP_M, out1 => "Line_Control_DB".Line[#Alm_REQ].Timers_Stop[5].SP_M)
      Move(in := "Line_Control_DB".Line[0].Timers_Stop[4].SP_S, out1 => "Line_Control_DB".Line[#Alm_REQ].Timers_Stop[4].SP_S)
      Move(in := "Line_Control_DB".Line[0].Timers_Stop[5].SP_S, out1 => "Line_Control_DB".Line[#Alm_REQ].Timers_Stop[5].SP_S)
   END_RUNG
   // the same network as SCL:
   IF #Ready THEN
       "Line_Control_DB".Line[#Alm_REQ].Timers_Stop[0].SP_M := "Line_Control_DB".Line[0].Timers_Stop[0].SP_M;
       "Line_Control_DB".Line[#Alm_REQ].Timers_Stop[1].SP_M := "Line_Control_DB".Line[0].Timers_Stop[1].SP_M;
       "Line_Control_DB".Line[#Alm_REQ].Timers_Stop[2].SP_M := "Line_Control_DB".Line[0].Timers_Stop[2].SP_M;
       "Line_Control_DB".Line[#Alm_REQ].Timers_Stop[3].SP_M := "Line_Control_DB".Line[0].Timers_Stop[3].SP_M;
       "Line_Control_DB".Line[#Alm_REQ].Timers_Stop[0].SP_S := "Line_Control_DB".Line[0].Timers_Stop[0].SP_S;
       "Line_Control_DB".Line[#Alm_REQ].Timers_Stop[1].SP_S := "Line_Control_DB".Line[0].Timers_Stop[1].SP_S;
       "Line_Control_DB".Line[#Alm_REQ].Timers_Stop[2].SP_S := "Line_Control_DB".Line[0].Timers_Stop[2].SP_S;
       "Line_Control_DB".Line[#Alm_REQ].Timers_Stop[3].SP_S := "Line_Control_DB".Line[0].Timers_Stop[3].SP_S;
       "Line_Control_DB".Line[#Alm_REQ].Timers_Stop[4].SP_M := "Line_Control_DB".Line[0].Timers_Stop[4].SP_M;
       "Line_Control_DB".Line[#Alm_REQ].Timers_Stop[5].SP_M := "Line_Control_DB".Line[0].Timers_Stop[5].SP_M;
       "Line_Control_DB".Line[#Alm_REQ].Timers_Stop[4].SP_S := "Line_Control_DB".Line[0].Timers_Stop[4].SP_S;
       "Line_Control_DB".Line[#Alm_REQ].Timers_Stop[5].SP_S := "Line_Control_DB".Line[0].Timers_Stop[5].SP_S;
   END_IF;
END_REGION

REGION Network 12: Чтение данных из выбранной линии в нулевой экземпляр для отображения на дисплее
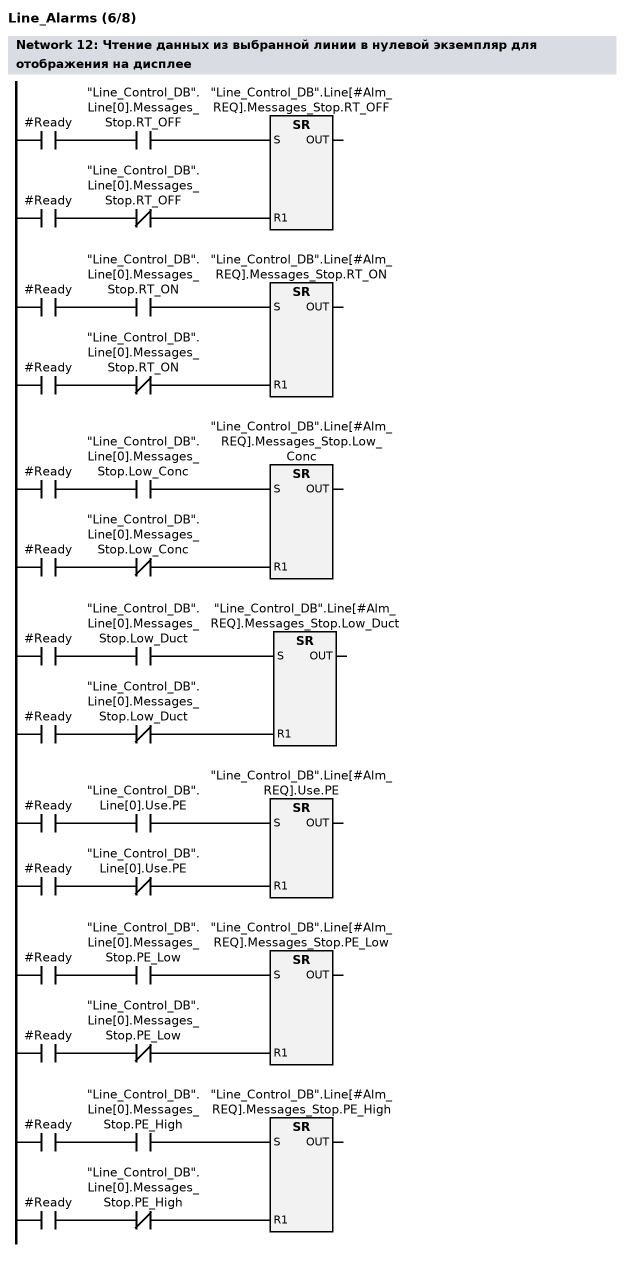
   RUNG wire#powerrail
      Contact( #Ready )
      Contact( "Line_Control_DB".Line[0].Messages_Stop.RT_OFF )
      S_SR(operand := "Line_Control_DB".Line[#Alm_REQ].Messages_Stop.RT_OFF, r1 := wire#w1)
   END_RUNG
   RUNG wire#powerrail
      Contact( #Ready )
      I_Contact( "Line_Control_DB".Line[0].Messages_Stop.RT_OFF )
   END_RUNG wire#w1
   RUNG wire#powerrail
      Contact( #Ready )
      Contact( "Line_Control_DB".Line[0].Messages_Stop.RT_ON )
      S_SR(operand := "Line_Control_DB".Line[#Alm_REQ].Messages_Stop.RT_ON, r1 := wire#w2)
   END_RUNG
   RUNG wire#powerrail
      Contact( #Ready )
      I_Contact( "Line_Control_DB".Line[0].Messages_Stop.RT_ON )
   END_RUNG wire#w2
   RUNG wire#powerrail
      Contact( #Ready )
      Contact( "Line_Control_DB".Line[0].Messages_Stop.Low_Conc )
      S_SR(operand := "Line_Control_DB".Line[#Alm_REQ].Messages_Stop.Low_Conc, r1 := wire#w3)
   END_RUNG
   RUNG wire#powerrail
      Contact( #Ready )
      I_Contact( "Line_Control_DB".Line[0].Messages_Stop.Low_Conc )
   END_RUNG wire#w3
   RUNG wire#powerrail
      Contact( #Ready )
      Contact( "Line_Control_DB".Line[0].Messages_Stop.Low_Duct )
      S_SR(operand := "Line_Control_DB".Line[#Alm_REQ].Messages_Stop.Low_Duct, r1 := wire#w4)
   END_RUNG
   RUNG wire#powerrail
      Contact( #Ready )
      I_Contact( "Line_Control_DB".Line[0].Messages_Stop.Low_Duct )
   END_RUNG wire#w4
   RUNG wire#powerrail
      Contact( #Ready )
      Contact( "Line_Control_DB".Line[0].Use.PE )
      S_SR(operand := "Line_Control_DB".Line[#Alm_REQ].Use.PE, r1 := wire#w5)
   END_RUNG
   RUNG wire#powerrail
      Contact( #Ready )
      I_Contact( "Line_Control_DB".Line[0].Use.PE )
   END_RUNG wire#w5
   RUNG wire#powerrail
      Contact( #Ready )
      Contact( "Line_Control_DB".Line[0].Messages_Stop.PE_Low )
      S_SR(operand := "Line_Control_DB".Line[#Alm_REQ].Messages_Stop.PE_Low, r1 := wire#w6)
   END_RUNG
   RUNG wire#powerrail
      Contact( #Ready )
      I_Contact( "Line_Control_DB".Line[0].Messages_Stop.PE_Low )
   END_RUNG wire#w6
   RUNG wire#powerrail
      Contact( #Ready )
      Contact( "Line_Control_DB".Line[0].Messages_Stop.PE_High )
      S_SR(operand := "Line_Control_DB".Line[#Alm_REQ].Messages_Stop.PE_High, r1 := wire#w7)
   END_RUNG
   RUNG wire#powerrail
      Contact( #Ready )
      I_Contact( "Line_Control_DB".Line[0].Messages_Stop.PE_High )
   END_RUNG wire#w7
   // the same network as SCL:
   #_w1 := #Ready AND NOT "Line_Control_DB".Line[0].Messages_Stop.RT_OFF;
   IF #Ready AND "Line_Control_DB".Line[0].Messages_Stop.RT_OFF THEN
       "Line_Control_DB".Line[#Alm_REQ].Messages_Stop.RT_OFF := TRUE;   // SR flip-flop
   END_IF;
   IF #_w1 THEN "Line_Control_DB".Line[#Alm_REQ].Messages_Stop.RT_OFF := FALSE; END_IF;
   #_w2 := #Ready AND NOT "Line_Control_DB".Line[0].Messages_Stop.RT_ON;
   IF #Ready AND "Line_Control_DB".Line[0].Messages_Stop.RT_ON THEN
       "Line_Control_DB".Line[#Alm_REQ].Messages_Stop.RT_ON := TRUE;   // SR flip-flop
   END_IF;
   IF #_w2 THEN "Line_Control_DB".Line[#Alm_REQ].Messages_Stop.RT_ON := FALSE; END_IF;
   #_w3 := #Ready AND NOT "Line_Control_DB".Line[0].Messages_Stop.Low_Conc;
   IF #Ready AND "Line_Control_DB".Line[0].Messages_Stop.Low_Conc THEN
       "Line_Control_DB".Line[#Alm_REQ].Messages_Stop.Low_Conc := TRUE;   // SR flip-flop
   END_IF;
   IF #_w3 THEN "Line_Control_DB".Line[#Alm_REQ].Messages_Stop.Low_Conc := FALSE; END_IF;
   #_w4 := #Ready AND NOT "Line_Control_DB".Line[0].Messages_Stop.Low_Duct;
   IF #Ready AND "Line_Control_DB".Line[0].Messages_Stop.Low_Duct THEN
       "Line_Control_DB".Line[#Alm_REQ].Messages_Stop.Low_Duct := TRUE;   // SR flip-flop
   END_IF;
   IF #_w4 THEN "Line_Control_DB".Line[#Alm_REQ].Messages_Stop.Low_Duct := FALSE; END_IF;
   #_w5 := #Ready AND NOT "Line_Control_DB".Line[0].Use.PE;
   IF #Ready AND "Line_Control_DB".Line[0].Use.PE THEN
       "Line_Control_DB".Line[#Alm_REQ].Use.PE := TRUE;   // SR flip-flop
   END_IF;
   IF #_w5 THEN "Line_Control_DB".Line[#Alm_REQ].Use.PE := FALSE; END_IF;
   #_w6 := #Ready AND NOT "Line_Control_DB".Line[0].Messages_Stop.PE_Low;
   IF #Ready AND "Line_Control_DB".Line[0].Messages_Stop.PE_Low THEN
       "Line_Control_DB".Line[#Alm_REQ].Messages_Stop.PE_Low := TRUE;   // SR flip-flop
   END_IF;
   IF #_w6 THEN "Line_Control_DB".Line[#Alm_REQ].Messages_Stop.PE_Low := FALSE; END_IF;
   #_w7 := #Ready AND NOT "Line_Control_DB".Line[0].Messages_Stop.PE_High;
   IF #Ready AND "Line_Control_DB".Line[0].Messages_Stop.PE_High THEN
       "Line_Control_DB".Line[#Alm_REQ].Messages_Stop.PE_High := TRUE;   // SR flip-flop
   END_IF;
   IF #_w7 THEN "Line_Control_DB".Line[#Alm_REQ].Messages_Stop.PE_High := FALSE; END_IF;
END_REGION

REGION Network 13: Чтение данных из выбранной линии в нулевой экземпляр для отображения на дисплее
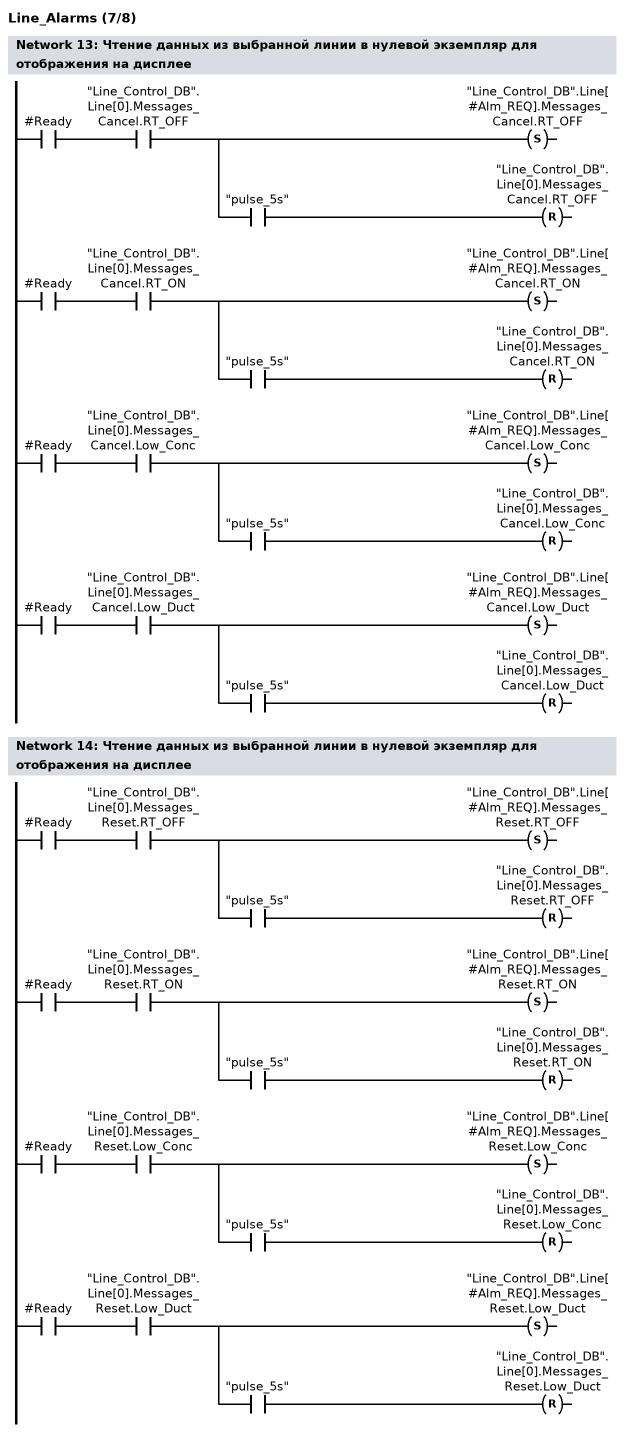
   RUNG wire#powerrail
      Contact( #Ready )
      Contact( "Line_Control_DB".Line[0].Messages_Cancel.RT_OFF )
      wire#w1
      S_Coil( "Line_Control_DB".Line[#Alm_REQ].Messages_Cancel.RT_OFF )
   END_RUNG
   RUNG wire#w1
      Contact( "pulse_5s" )
      R_Coil( "Line_Control_DB".Line[0].Messages_Cancel.RT_OFF )
   END_RUNG
   RUNG wire#powerrail
      Contact( #Ready )
      Contact( "Line_Control_DB".Line[0].Messages_Cancel.RT_ON )
      wire#w2
      S_Coil( "Line_Control_DB".Line[#Alm_REQ].Messages_Cancel.RT_ON )
   END_RUNG
   RUNG wire#w2
      Contact( "pulse_5s" )
      R_Coil( "Line_Control_DB".Line[0].Messages_Cancel.RT_ON )
   END_RUNG
   RUNG wire#powerrail
      Contact( #Ready )
      Contact( "Line_Control_DB".Line[0].Messages_Cancel.Low_Conc )
      wire#w3
      S_Coil( "Line_Control_DB".Line[#Alm_REQ].Messages_Cancel.Low_Conc )
   END_RUNG
   RUNG wire#w3
      Contact( "pulse_5s" )
      R_Coil( "Line_Control_DB".Line[0].Messages_Cancel.Low_Conc )
   END_RUNG
   RUNG wire#powerrail
      Contact( #Ready )
      Contact( "Line_Control_DB".Line[0].Messages_Cancel.Low_Duct )
      wire#w4
      S_Coil( "Line_Control_DB".Line[#Alm_REQ].Messages_Cancel.Low_Duct )
   END_RUNG
   RUNG wire#w4
      Contact( "pulse_5s" )
      R_Coil( "Line_Control_DB".Line[0].Messages_Cancel.Low_Duct )
   END_RUNG
   // the same network as SCL:
   #_w1 := #Ready AND "Line_Control_DB".Line[0].Messages_Cancel.RT_OFF;
   IF #_w1 THEN "Line_Control_DB".Line[#Alm_REQ].Messages_Cancel.RT_OFF := TRUE; END_IF;
   IF #_w1 AND "pulse_5s" THEN "Line_Control_DB".Line[0].Messages_Cancel.RT_OFF := FALSE; END_IF;
   #_w2 := #Ready AND "Line_Control_DB".Line[0].Messages_Cancel.RT_ON;
   IF #_w2 THEN "Line_Control_DB".Line[#Alm_REQ].Messages_Cancel.RT_ON := TRUE; END_IF;
   IF #_w2 AND "pulse_5s" THEN "Line_Control_DB".Line[0].Messages_Cancel.RT_ON := FALSE; END_IF;
   #_w3 := #Ready AND "Line_Control_DB".Line[0].Messages_Cancel.Low_Conc;
   IF #_w3 THEN "Line_Control_DB".Line[#Alm_REQ].Messages_Cancel.Low_Conc := TRUE; END_IF;
   IF #_w3 AND "pulse_5s" THEN "Line_Control_DB".Line[0].Messages_Cancel.Low_Conc := FALSE; END_IF;
   #_w4 := #Ready AND "Line_Control_DB".Line[0].Messages_Cancel.Low_Duct;
   IF #_w4 THEN "Line_Control_DB".Line[#Alm_REQ].Messages_Cancel.Low_Duct := TRUE; END_IF;
   IF #_w4 AND "pulse_5s" THEN "Line_Control_DB".Line[0].Messages_Cancel.Low_Duct := FALSE; END_IF;
END_REGION

REGION Network 14: Чтение данных из выбранной линии в нулевой экземпляр для отображения на дисплее
   RUNG wire#powerrail
      Contact( #Ready )
      Contact( "Line_Control_DB".Line[0].Messages_Reset.RT_OFF )
      wire#w1
      S_Coil( "Line_Control_DB".Line[#Alm_REQ].Messages_Reset.RT_OFF )
   END_RUNG
   RUNG wire#w1
      Contact( "pulse_5s" )
      R_Coil( "Line_Control_DB".Line[0].Messages_Reset.RT_OFF )
   END_RUNG
   RUNG wire#powerrail
      Contact( #Ready )
      Contact( "Line_Control_DB".Line[0].Messages_Reset.RT_ON )
      wire#w2
      S_Coil( "Line_Control_DB".Line[#Alm_REQ].Messages_Reset.RT_ON )
   END_RUNG
   RUNG wire#w2
      Contact( "pulse_5s" )
      R_Coil( "Line_Control_DB".Line[0].Messages_Reset.RT_ON )
   END_RUNG
   RUNG wire#powerrail
      Contact( #Ready )
      Contact( "Line_Control_DB".Line[0].Messages_Reset.Low_Conc )
      wire#w3
      S_Coil( "Line_Control_DB".Line[#Alm_REQ].Messages_Reset.Low_Conc )
   END_RUNG
   RUNG wire#w3
      Contact( "pulse_5s" )
      R_Coil( "Line_Control_DB".Line[0].Messages_Reset.Low_Conc )
   END_RUNG
   RUNG wire#powerrail
      Contact( #Ready )
      Contact( "Line_Control_DB".Line[0].Messages_Reset.Low_Duct )
      wire#w4
      S_Coil( "Line_Control_DB".Line[#Alm_REQ].Messages_Reset.Low_Duct )
   END_RUNG
   RUNG wire#w4
      Contact( "pulse_5s" )
      R_Coil( "Line_Control_DB".Line[0].Messages_Reset.Low_Duct )
   END_RUNG
   // the same network as SCL:
   #_w1 := #Ready AND "Line_Control_DB".Line[0].Messages_Reset.RT_OFF;
   IF #_w1 THEN "Line_Control_DB".Line[#Alm_REQ].Messages_Reset.RT_OFF := TRUE; END_IF;
   IF #_w1 AND "pulse_5s" THEN "Line_Control_DB".Line[0].Messages_Reset.RT_OFF := FALSE; END_IF;
   #_w2 := #Ready AND "Line_Control_DB".Line[0].Messages_Reset.RT_ON;
   IF #_w2 THEN "Line_Control_DB".Line[#Alm_REQ].Messages_Reset.RT_ON := TRUE; END_IF;
   IF #_w2 AND "pulse_5s" THEN "Line_Control_DB".Line[0].Messages_Reset.RT_ON := FALSE; END_IF;
   #_w3 := #Ready AND "Line_Control_DB".Line[0].Messages_Reset.Low_Conc;
   IF #_w3 THEN "Line_Control_DB".Line[#Alm_REQ].Messages_Reset.Low_Conc := TRUE; END_IF;
   IF #_w3 AND "pulse_5s" THEN "Line_Control_DB".Line[0].Messages_Reset.Low_Conc := FALSE; END_IF;
   #_w4 := #Ready AND "Line_Control_DB".Line[0].Messages_Reset.Low_Duct;
   IF #_w4 THEN "Line_Control_DB".Line[#Alm_REQ].Messages_Reset.Low_Duct := TRUE; END_IF;
   IF #_w4 AND "pulse_5s" THEN "Line_Control_DB".Line[0].Messages_Reset.Low_Duct := FALSE; END_IF;
END_REGION

REGION Network 15: Чтение данных из выбранной линии в нулевой экземпляр для отображения на дисплее
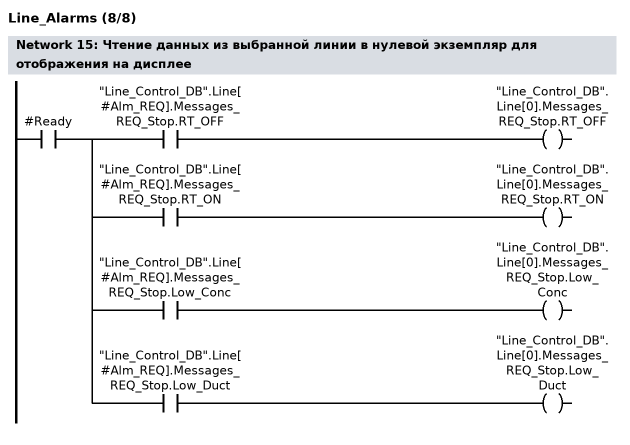
   RUNG wire#powerrail
      Contact( #Ready )
      wire#w1
      Contact( "Line_Control_DB".Line[#Alm_REQ].Messages_REQ_Stop.RT_OFF )
      Coil( "Line_Control_DB".Line[0].Messages_REQ_Stop.RT_OFF )
   END_RUNG
   RUNG wire#w1
      Contact( "Line_Control_DB".Line[#Alm_REQ].Messages_REQ_Stop.RT_ON )
      Coil( "Line_Control_DB".Line[0].Messages_REQ_Stop.RT_ON )
   END_RUNG
   RUNG wire#w1
      Contact( "Line_Control_DB".Line[#Alm_REQ].Messages_REQ_Stop.Low_Conc )
      Coil( "Line_Control_DB".Line[0].Messages_REQ_Stop.Low_Conc )
   END_RUNG
   RUNG wire#w1
      Contact( "Line_Control_DB".Line[#Alm_REQ].Messages_REQ_Stop.Low_Duct )
      Coil( "Line_Control_DB".Line[0].Messages_REQ_Stop.Low_Duct )
   END_RUNG
   // the same network as SCL:
   "Line_Control_DB".Line[0].Messages_REQ_Stop.RT_OFF := #Ready AND "Line_Control_DB".Line[#Alm_REQ].Messages_REQ_Stop.RT_OFF;
   "Line_Control_DB".Line[0].Messages_REQ_Stop.RT_ON := #Ready AND "Line_Control_DB".Line[#Alm_REQ].Messages_REQ_Stop.RT_ON;
   "Line_Control_DB".Line[0].Messages_REQ_Stop.Low_Conc := #Ready AND "Line_Control_DB".Line[#Alm_REQ].Messages_REQ_Stop.Low_Conc;
   "Line_Control_DB".Line[0].Messages_REQ_Stop.Low_Duct := #Ready AND "Line_Control_DB".Line[#Alm_REQ].Messages_REQ_Stop.Low_Duct;
END_REGION
END_FUNCTION
